// TIA Portal V17 export
// export: Created 2025-03-20T13:42:25.2764009Z, ExportSetting WithDefaults, DisplayName Totally Integrated Automation Portal, DisplayVersion V17 Update 8, DisplayName TIA Portal Openness, DisplayVersion V17 Update 8, DisplayName TIA Portal Version Control Interface, DisplayVersion V17, DisplayName SINAMICS Startdrive Advanced, DisplayVersion V17 SP2, DisplayName SINAMICS Startdrive G110M, G120, G120C, G120D, G120P, G115D, DisplayVersion V17 SP2, DisplayName SINAMICS Startdrive G130, G150, S120, S150, SINAMICS MV, S210, DisplayVersion V17 SP2, DisplayName STEP 7 Professional, DisplayVersion V17 Update 8, DisplayName SINUMERIK ONE STEP 7 Toolbox, DisplayVersion V17 Update 12, DisplayName SINUMERIK 840D sl STEP 7 Toolbox, DisplayVersion V17 Update 12, DisplayName STEP 7 Safety, DisplayVersion V17 Update 6, DisplayName WinCC Advanced, DisplayVersion V17 Update 8
FUNCTION_BLOCK "FB22501_TEMPERATURE_JKT_CONTROL"   // FB22501, LAD
TITLE = FB22501 TEMPERATURE JKT CONTROL
{ S7_Optimized_Access := 'FALSE' }
VERSION : 0.1
// stored: AutoNumber false, IsIECCheckEnabled false, SetENOAutomatically false, UDAEnableTagReadback false
   VAR_INPUT
      iFEEDBACK_TEMP : Real;
      iCONTROL_ON_DELAYED : Bool;
      iBREAKER : Bool;
      iMANUAL_START_REQUEST : Bool;
      iMANUAL_STOP_REQUEST : Bool;
   END_VAR
   VAR_OUTPUT
      oANALOG_TEMP_VALUE : Int;
      oSwitchoncondition_on : Bool;
   END_VAR
   VAR DB_SPECIFIC
      DATA : Struct
         Start : Bool;
         Conditions : Bool;
         "Auto Cons." : Real;
         Consignment : Real;
         Min_Range : Real;
         Max_Range : Real;
         Lim_Lo : Real;
         Lim_HI : Real;
         "HMI Manual Cons." : Real;
         "HMI Feedback Value" : Real;
         "HMI Consignment" : Real;
      END_STRUCT;
   END_VAR
   VAR_TEMP
      RetVal : Int;
      TmpNormal : Real;
   END_VAR
   VAR_TEMP   // added for the SCL form of the ladder/FBD networks
      _w1 : Bool;
   END_VAR
BEGIN

REGION Network 1: CONDITIONS / Conditions
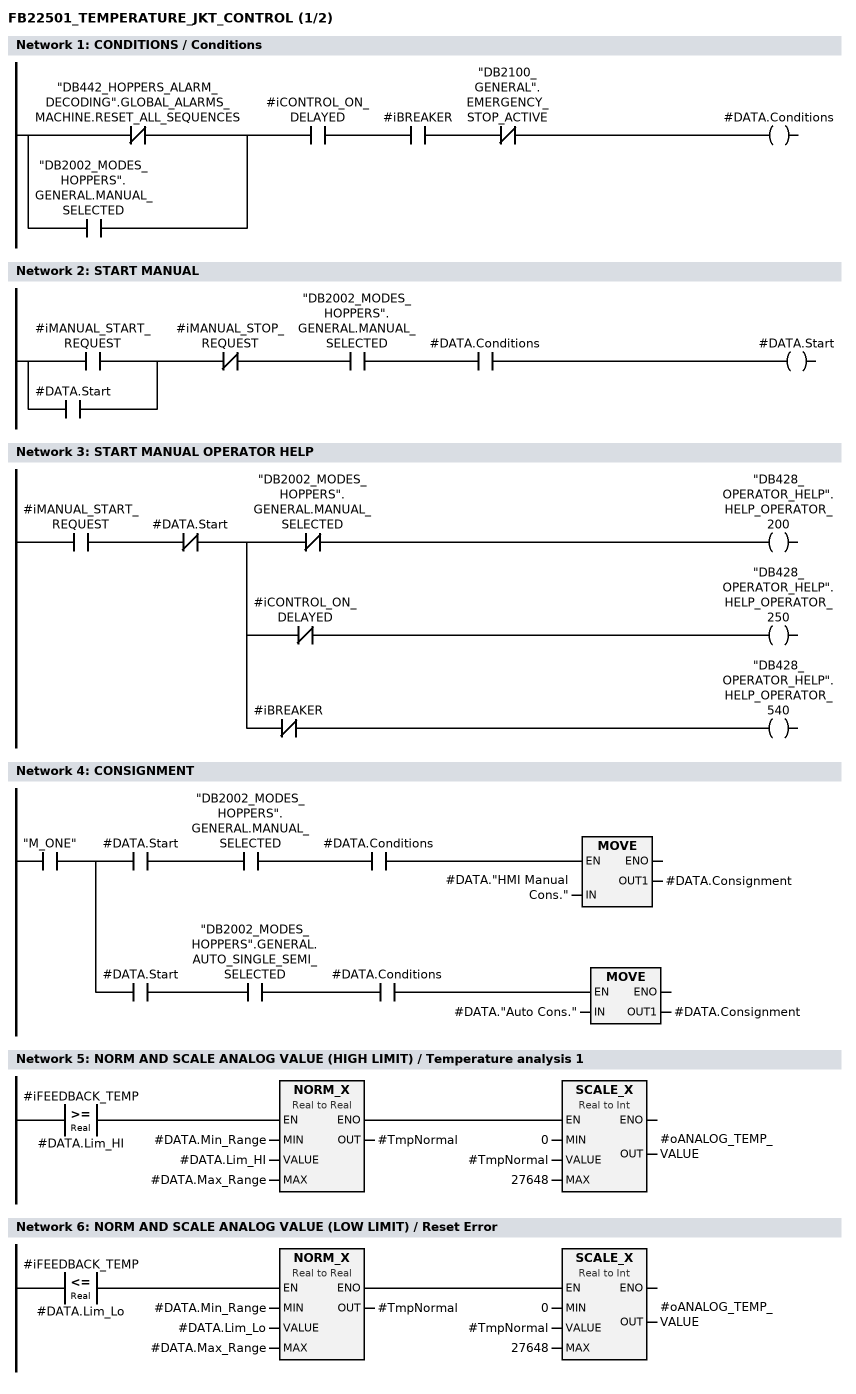
   RUNG wire#powerrail
      I_Contact( "DB442_HOPPERS_ALARM_DECODING".GLOBAL_ALARMS_MACHINE.RESET_ALL_SEQUENCES )
      wire#w1
      Contact( #iCONTROL_ON_DELAYED )
      Contact( #iBREAKER )
      I_Contact( "DB2100_GENERAL".EMERGENCY_STOP_ACTIVE )
      Coil( #DATA.Conditions )
   END_RUNG
   RUNG wire#powerrail
      Contact( "DB2002_MODES_HOPPERS".GENERAL.MANUAL_SELECTED )
   END_RUNG wire#w1
   // the same network as SCL:
   #DATA.Conditions := (NOT "DB442_HOPPERS_ALARM_DECODING".GLOBAL_ALARMS_MACHINE.RESET_ALL_SEQUENCES OR "DB2002_MODES_HOPPERS".GENERAL.MANUAL_SELECTED) AND #iCONTROL_ON_DELAYED AND #iBREAKER AND NOT "DB2100_GENERAL".EMERGENCY_STOP_ACTIVE;
END_REGION

REGION Network 2: START MANUAL
   RUNG wire#powerrail
      Contact( #iMANUAL_START_REQUEST )
      wire#w1
      I_Contact( #iMANUAL_STOP_REQUEST )
      Contact( "DB2002_MODES_HOPPERS".GENERAL.MANUAL_SELECTED )
      Contact( #DATA.Conditions )
      Coil( #DATA.Start )
   END_RUNG
   RUNG wire#powerrail
      Contact( #DATA.Start )
   END_RUNG wire#w1
   // the same network as SCL:
   #DATA.Start := (#iMANUAL_START_REQUEST OR #DATA.Start) AND NOT #iMANUAL_STOP_REQUEST AND "DB2002_MODES_HOPPERS".GENERAL.MANUAL_SELECTED AND #DATA.Conditions;
END_REGION

REGION Network 3: START MANUAL OPERATOR HELP
   RUNG wire#powerrail
      Contact( #iMANUAL_START_REQUEST )
      I_Contact( #DATA.Start )
      wire#w1
      I_Contact( "DB2002_MODES_HOPPERS".GENERAL.MANUAL_SELECTED )
      Coil( "DB428_OPERATOR_HELP".HELP_OPERATOR_200 )
   END_RUNG
   RUNG wire#w1
      I_Contact( #iCONTROL_ON_DELAYED )
      Coil( "DB428_OPERATOR_HELP".HELP_OPERATOR_250 )
   END_RUNG
   RUNG wire#w1
      I_Contact( #iBREAKER )
      Coil( "DB428_OPERATOR_HELP".HELP_OPERATOR_540 )
   END_RUNG
   // the same network as SCL:
   #_w1 := #iMANUAL_START_REQUEST AND NOT #DATA.Start;
   "DB428_OPERATOR_HELP".HELP_OPERATOR_200 := #_w1 AND NOT "DB2002_MODES_HOPPERS".GENERAL.MANUAL_SELECTED;
   "DB428_OPERATOR_HELP".HELP_OPERATOR_250 := #_w1 AND NOT #iCONTROL_ON_DELAYED;
   "DB428_OPERATOR_HELP".HELP_OPERATOR_540 := #_w1 AND NOT #iBREAKER;
END_REGION

REGION Network 4: CONSIGNMENT
   RUNG wire#powerrail
      Contact( "M_ONE" )
      wire#w1
      Contact( #DATA.Start )
      Contact( "DB2002_MODES_HOPPERS".GENERAL.MANUAL_SELECTED )
      Contact( #DATA.Conditions )
      Move(in := #DATA."HMI Manual Cons.", out1 => #DATA.Consignment)
   END_RUNG
   RUNG wire#w1
      Contact( #DATA.Start )
      Contact( "DB2002_MODES_HOPPERS".GENERAL.AUTO_SINGLE_SEMI_SELECTED )
      Contact( #DATA.Conditions )
      Move(in := #DATA."Auto Cons.", out1 => #DATA.Consignment)
   END_RUNG
   // the same network as SCL:
   IF "M_ONE" AND #DATA.Start AND "DB2002_MODES_HOPPERS".GENERAL.MANUAL_SELECTED AND #DATA.Conditions THEN
       #DATA.Consignment := #DATA."HMI Manual Cons.";
   END_IF;
   IF "M_ONE" AND #DATA.Start AND "DB2002_MODES_HOPPERS".GENERAL.AUTO_SINGLE_SEMI_SELECTED AND #DATA.Conditions THEN
       #DATA.Consignment := #DATA."Auto Cons.";
   END_IF;
END_REGION

REGION Network 5: NORM AND SCALE ANALOG VALUE (HIGH LIMIT) / Temperature analysis 1
   RUNG wire#powerrail
      { S7_Templates := "SrcType := Real" } GE_Contact(in1 := #iFEEDBACK_TEMP, in2 := #DATA.Lim_HI)
      { S7_Templates := "[SrcType := Real, DestType := Real]" } Normalize(min := #DATA.Min_Range, value := #DATA.Lim_HI, max := #DATA.Max_Range, out => #TmpNormal)
      { S7_Templates := "[SrcType := Real, DestType := Int]" } Scale(min := 0, value := #TmpNormal, max := 27648, out => #oANALOG_TEMP_VALUE)
   END_RUNG
   // the same network as SCL:
   IF #iFEEDBACK_TEMP >= #DATA.Lim_HI THEN
       #TmpNormal := NORM_X(MIN := #DATA.Min_Range, VALUE := #DATA.Lim_HI, MAX := #DATA.Max_Range);
       #oANALOG_TEMP_VALUE := SCALE_X(MIN := 0, VALUE := #TmpNormal, MAX := 27648);
   END_IF;
END_REGION

REGION Network 6: NORM AND SCALE ANALOG VALUE (LOW LIMIT) / Reset Error
   RUNG wire#powerrail
      { S7_Templates := "SrcType := Real" } LE_Contact(in1 := #iFEEDBACK_TEMP, in2 := #DATA.Lim_Lo)
      { S7_Templates := "[SrcType := Real, DestType := Real]" } Normalize(min := #DATA.Min_Range, value := #DATA.Lim_Lo, max := #DATA.Max_Range, out => #TmpNormal)
      { S7_Templates := "[SrcType := Real, DestType := Int]" } Scale(min := 0, value := #TmpNormal, max := 27648, out => #oANALOG_TEMP_VALUE)
   END_RUNG
   // the same network as SCL:
   IF #iFEEDBACK_TEMP <= #DATA.Lim_Lo THEN
       #TmpNormal := NORM_X(MIN := #DATA.Min_Range, VALUE := #DATA.Lim_Lo, MAX := #DATA.Max_Range);
       #oANALOG_TEMP_VALUE := SCALE_X(MIN := 0, VALUE := #TmpNormal, MAX := 27648);
   END_IF;
END_REGION

REGION Network 7: NORM AND SCALE ANALOG VALUE / Scale to analog value / Cooling water flow
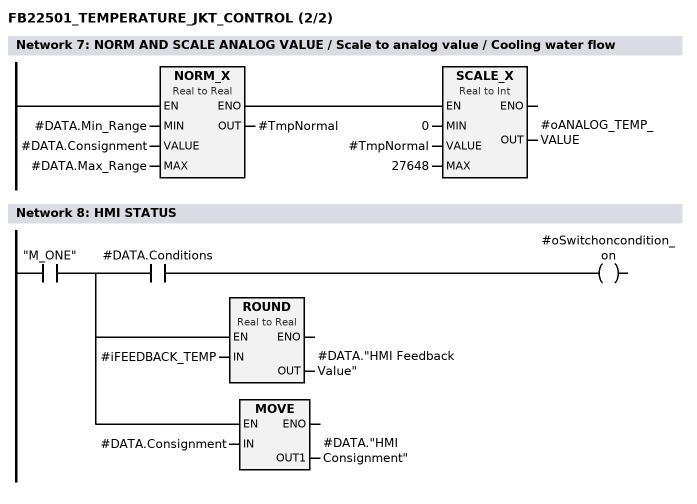
   RUNG wire#powerrail
      { S7_Templates := "[SrcType := Real, DestType := Real]" } Normalize(min := #DATA.Min_Range, value := #DATA.Consignment, max := #DATA.Max_Range, out => #TmpNormal)
      { S7_Templates := "[SrcType := Real, DestType := Int]" } Scale(min := 0, value := #TmpNormal, max := 27648, out => #oANALOG_TEMP_VALUE)
   END_RUNG
   // the same network as SCL:
   #TmpNormal := NORM_X(MIN := #DATA.Min_Range, VALUE := #DATA.Consignment, MAX := #DATA.Max_Range);
   #oANALOG_TEMP_VALUE := SCALE_X(MIN := 0, VALUE := #TmpNormal, MAX := 27648);
END_REGION

REGION Network 8: HMI STATUS
   RUNG wire#powerrail
      Contact( "M_ONE" )
      wire#w1
      Contact( #DATA.Conditions )
      Coil( #oSwitchoncondition_on )
   END_RUNG
   RUNG wire#w1
      { S7_Templates := "[SrcType := Real, DestType := Real]" } Round(in := #iFEEDBACK_TEMP, out => #DATA."HMI Feedback Value")
   END_RUNG
   RUNG wire#w1
      Move(in := #DATA.Consignment, out1 => #DATA."HMI Consignment")
   END_RUNG
   // the same network as SCL:
   #oSwitchoncondition_on := "M_ONE" AND #DATA.Conditions;
   IF "M_ONE" THEN
       #DATA."HMI Feedback Value" := ROUND(#iFEEDBACK_TEMP);
       #DATA."HMI Consignment" := #DATA.Consignment;
   END_IF;
END_REGION
END_FUNCTION_BLOCK
